(* Logix 5000 project; controller Laser_Cutter vendor 1 type 14 code 149 rev 28.11; software revision 28.00; part 3 of 4 *)
(* tags used below, declared in another part *)
   aDoorSafetySwitchUnlockSol : BOOL;
   aExhaustStart : BOOL;
   alarmActive : BOOL;
   aTapForward : BOOL;
   aTapReverse : BOOL;
   automaticSeqStep : DINT;
   autoMode : BOOL;
   autoModeReady : BOOL;
   boltDriverDownDB : TIMER;
   boltDriverUpDB : TIMER;
   boltPresentAtInfeedDB : TIMER;
   clampStation2DB : TIMER;
   clampStation4DB : TIMER;
   clampStation5DB : TIMER;
   collarAtStation1DB : TIMER;
   collarAtStation2DB : TIMER;
   collarAtStation3DB : TIMER;
   collarAtStation4DB : TIMER;
   collarAtStation5DB : TIMER;
   collarFeedingTrackHighLevelDB : TIMER;
   collarFeedingTrackLowLevelDB : TIMER;
   collarPresentAtInfeedDB : TIMER;
   Counter : DINT;
   Counter2 : DINT;
   Counter3 : DINT;
   CYCLE_IN_PROG : BOOL;
   cycleComplete : BOOL;
   doorClosedDebounceTimer : TIMER;
   doorLockedDebounceTimer : TIMER;
   doorUnlockedDebounceTimer : TIMER;
   Exec_Laser_SR : BOOL;
   Exec_Robot_SR : BOOL;
   Exec_Tapping_SR : BOOL;
   execLoadPalletSR : BOOL;
   Execute_MoveToZoneSR : BOOL;
   Execute_RejectSR : BOOL;
   executeInitializationSequence : BOOL;
   hmiMessageNumber : DINT;
   hmiMessageNumberBuffer : DINT;
   hmiMessageString : STRING;
   hmiMessageStringArray : STRING[64];
   INIT_IN_PROG : BOOL;
   initHMIMessageDelayTimer : TIMER;
   initSeqStep : DINT;
   initTimeout : TIMER;
   LaserSeqStep : INT;
   loadPalletSeqStep : INT;
   manualMode : BOOL;
   MoveToZoneSeqStep : INT;
   mSecPulseOffTmr1 : TIMER;
   mSecPulseOnTmr1 : TIMER;
   oneSecPulseOffTmr : TIMER;
   oneSecPulseOnTmr : TIMER;
   palletShotpinRetractedDebounceTimer : TIMER;
   partsPresentDurringInitialization : BOOL;
   performOpControl : CONTROL;
   performOperation : DINT[1];
   rejectPartFlag : BOOL;
   rejectSeqStep : DINT;
   rejectShuttleAtAcceptDB : TIMER;
   rejectShuttleAtRejectDB : TIMER;
   remotePVDisplayNum : DINT;
   robotAtDropAPR : BOOL;
   robotAtHome : BOOL;
   robotAtPickAPR : BOOL;
   robotFinishedDrop : BOOL;
   robotHasBolt : BOOL;
   robotInMotion : BOOL;
   robotPickBolt : BOOL;
   robotScrewInBolt : BOOL;
   robotSeqStep : DINT;
   sendRobotToDropAPR : BOOL;
   sendRobotToHome : BOOL;
   sendRobotToPick : BOOL;
   startRobotSequence : BOOL;
   systemInInitializedPosition : BOOL;
   tapDownDB : TIMER;
   tapDwellTimer : TIMER;
   tapSeqStep : DINT;
   tapUpDB : TIMER;
   unclampStation2DB : TIMER;
   unclampStation4DB : TIMER;
   unclampStation5DB : TIMER;
   walkingBeamDownDB : TIMER;
   walkingBeamLeftDB : TIMER;
   walkingBeamRightDB : TIMER;
   walkingBeamUpDB : TIMER;
   boltDriverDown : ALIAS FOR MURR_IMPACT_IO_1:I.Data[1].6;
   boltDriverUp : ALIAS FOR MURR_IMPACT_IO_1:I.Data[1].5;
   boltPresentAtInfeed : ALIAS FOR MURR_IMPACT_IO_1:I.Data[0].5;
   cameraGoodPart : ALIAS FOR Local:1:I.Data.7;
   cameraOnline : ALIAS FOR Local:1:I.Data.9;
   clampStation2 : ALIAS FOR MURR_IMPACT_IO_1:I.Data[1].7;
   clampStation4 : ALIAS FOR MURR_IMPACT_IO_1:I.Data[2].1;
   clampStation5 : ALIAS FOR MURR_IMPACT_IO_1:I.Data[2].3;
   collarAtStation1 : ALIAS FOR MURR_IMPACT_IO_1:I.Data[0].6;
   collarAtStation2 : ALIAS FOR MURR_IMPACT_IO_1:I.Data[0].7;
   collarAtStation3 : ALIAS FOR MURR_IMPACT_IO_1:I.Data[1].0;
   collarAtStation4 : ALIAS FOR MURR_IMPACT_IO_1:I.Data[1].1;
   collarAtStation5 : ALIAS FOR MURR_IMPACT_IO_1:I.Data[1].2;
   collarFeedingTrackHighLevel : ALIAS FOR MURR_IMPACT_IO_1:I.Data[0].1;
   collarFeedingTrackLowLevel : ALIAS FOR MURR_IMPACT_IO_1:I.Data[0].0;
   collarPresentAtInfeed : ALIAS FOR MURR_IMPACT_IO_1:I.Data[0].4;
   currentUser : DINT;   // Access Level of current user
   doorOpenedSafetyRelayStatus : ALIAS FOR Local:1:I.Data.1;
   doorSafetySwitchUnlockSol : ALIAS FOR Local:1:O.Data.10;
   eStopSafetyRelayStatus : ALIAS FOR Local:1:I.Data.0;
   Local1IData10 : ALIAS FOR Local:1:I.Data.10;
   Local1IData11 : ALIAS FOR Local:1:I.Data.11;
   rejectShuttleAtAccept : ALIAS FOR MURR_IMPACT_IO_1:I.Data[2].5;
   rejectShuttleAtReject : ALIAS FOR MURR_IMPACT_IO_1:I.Data[2].6;
   stopPB : ALIAS FOR Local:1:I.Data.4;
   tapDown : ALIAS FOR MURR_IMPACT_IO_1:I.Data[1].4;
   tapUp : ALIAS FOR MURR_IMPACT_IO_1:I.Data[1].3;
   TO_DRV1 : CON_EIP_IN;
   TO_DRV2 : CON_EIP_IN;
   unclampStation2 : ALIAS FOR MURR_IMPACT_IO_1:I.Data[2].0;
   unclampStation4 : ALIAS FOR MURR_IMPACT_IO_1:I.Data[2].2;
   unclampStation5 : ALIAS FOR MURR_IMPACT_IO_1:I.Data[2].4;
   walkingBeamDown : ALIAS FOR MURR_IMPACT_IO_2:I.Data[0].0;
   walkingBeamLeft : ALIAS FOR MURR_IMPACT_IO_2:I.Data[0].2;
   walkingBeamRight : ALIAS FOR MURR_IMPACT_IO_2:I.Data[0].1;
   walkingBeamUp : ALIAS FOR MURR_IMPACT_IO_1:I.Data[2].7;
(* MainProgram, continued *)

ROUTINE Exec_Reject_SR   (* ladder *)
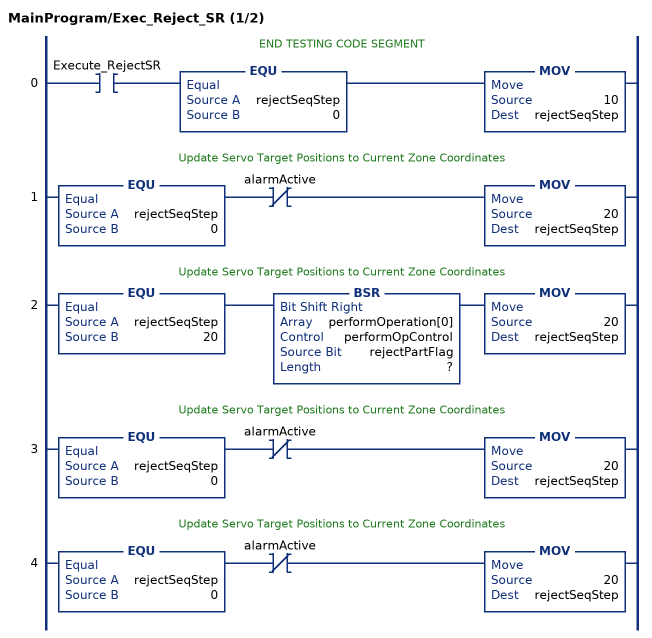
   // END TESTING CODE SEGMENT
   0: XIC(Execute_RejectSR)EQU(rejectSeqStep,0)MOV(10,rejectSeqStep);
   // Update Servo Target Positions to Current Zone Coordinates
   1: EQU(rejectSeqStep,0)XIO(alarmActive)MOV(20,rejectSeqStep);
   // Update Servo Target Positions to Current Zone Coordinates
   2: EQU(rejectSeqStep,20)BSR(performOperation[0],performOpControl,rejectPartFlag,?)MOV(20,rejectSeqStep);
   // Update Servo Target Positions to Current Zone Coordinates
   3: EQU(rejectSeqStep,0)XIO(alarmActive)MOV(20,rejectSeqStep);
   // Update Servo Target Positions to Current Zone Coordinates
   4: EQU(rejectSeqStep,0)XIO(alarmActive)MOV(20,rejectSeqStep);
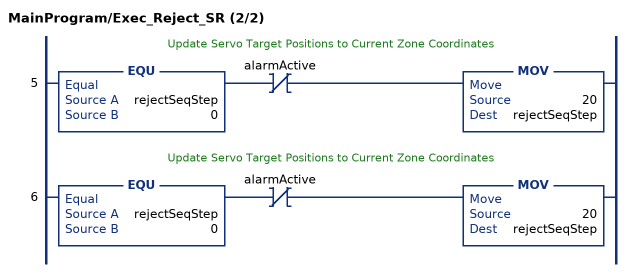
   // Update Servo Target Positions to Current Zone Coordinates
   5: EQU(rejectSeqStep,0)XIO(alarmActive)MOV(20,rejectSeqStep);
   // Update Servo Target Positions to Current Zone Coordinates
   6: EQU(rejectSeqStep,0)XIO(alarmActive)MOV(20,rejectSeqStep);
END_ROUTINE

ROUTINE Exec_Robot_SR   (* ladder *)
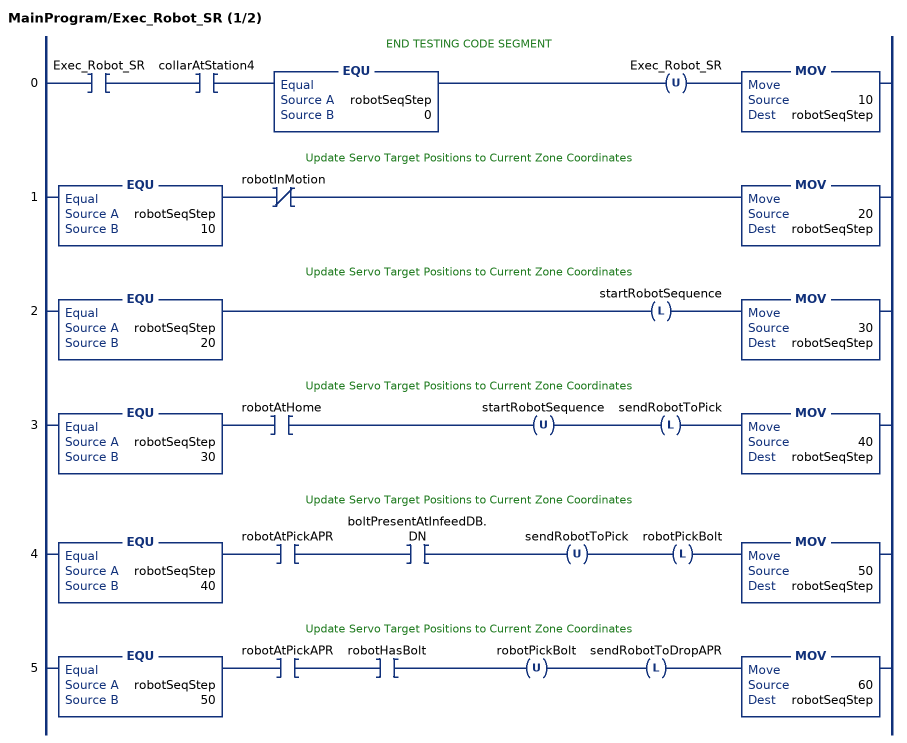
   // END TESTING CODE SEGMENT
   0: XIC(Exec_Robot_SR)XIC(collarAtStation4)EQU(robotSeqStep,0)OTU(Exec_Robot_SR)MOV(10,robotSeqStep);
   // Update Servo Target Positions to Current Zone Coordinates
   1: EQU(robotSeqStep,10)XIO(robotInMotion)MOV(20,robotSeqStep);
   // Update Servo Target Positions to Current Zone Coordinates
   2: EQU(robotSeqStep,20)OTL(startRobotSequence)MOV(30,robotSeqStep);
   // Update Servo Target Positions to Current Zone Coordinates
   3: EQU(robotSeqStep,30)XIC(robotAtHome)OTU(startRobotSequence)OTL(sendRobotToPick)MOV(40,robotSeqStep);
   // Update Servo Target Positions to Current Zone Coordinates
   4: EQU(robotSeqStep,40)XIC(robotAtPickAPR)XIC(boltPresentAtInfeedDB.DN)OTU(sendRobotToPick)OTL(robotPickBolt)MOV(50,robotSeqStep);
   // Update Servo Target Positions to Current Zone Coordinates
   5: EQU(robotSeqStep,50)XIC(robotAtPickAPR)XIC(robotHasBolt)OTU(robotPickBolt)OTL(sendRobotToDropAPR)MOV(60,robotSeqStep);
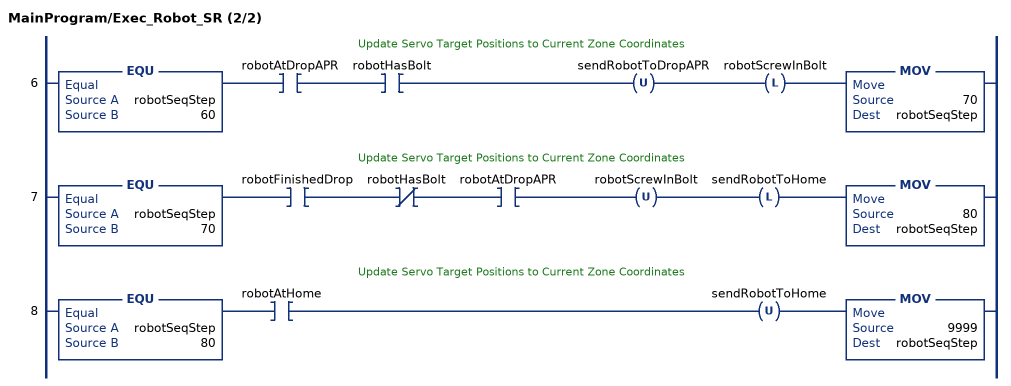
   // Update Servo Target Positions to Current Zone Coordinates
   6: EQU(robotSeqStep,60)XIC(robotAtDropAPR)XIC(robotHasBolt)OTU(sendRobotToDropAPR)OTL(robotScrewInBolt)MOV(70,robotSeqStep);
   // Update Servo Target Positions to Current Zone Coordinates
   7: EQU(robotSeqStep,70)XIC(robotFinishedDrop)XIO(robotHasBolt)XIC(robotAtDropAPR)OTU(robotScrewInBolt)OTL(sendRobotToHome)MOV(80,robotSeqStep);
   // Update Servo Target Positions to Current Zone Coordinates
   8: EQU(robotSeqStep,80)XIC(robotAtHome)OTU(sendRobotToHome)MOV(9999,robotSeqStep);
END_ROUTINE

ROUTINE Exec_Tapping_SR   (* ladder *)
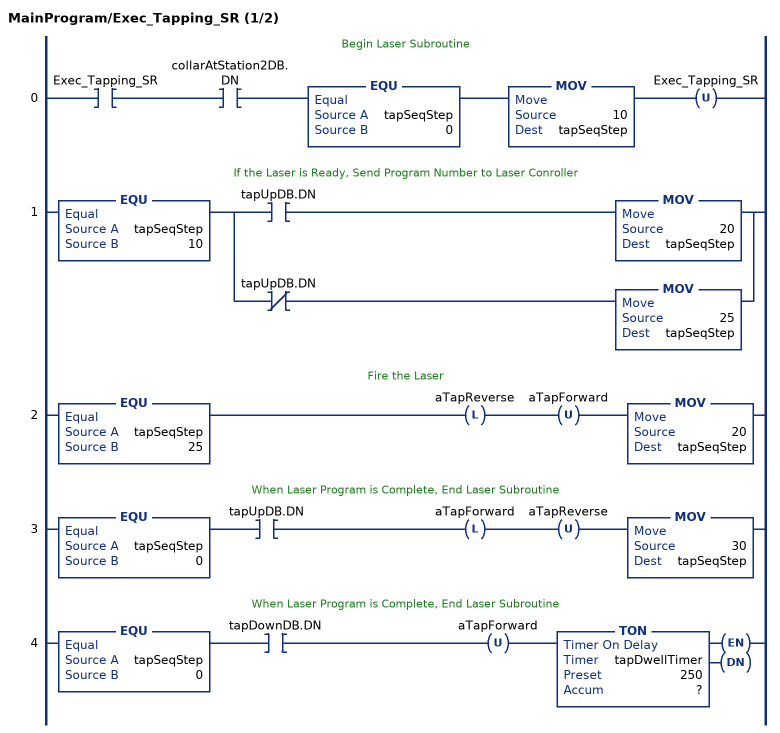
   // Begin Laser Subroutine
   0: XIC(Exec_Tapping_SR)XIC(collarAtStation2DB.DN)EQU(tapSeqStep,0)MOV(10,tapSeqStep)OTU(Exec_Tapping_SR);
   // If the Laser is Ready, Send Program Number to Laser Conroller
   1: EQU(tapSeqStep,10)[XIC(tapUpDB.DN) MOV(20,tapSeqStep) ,XIO(tapUpDB.DN) MOV(25,tapSeqStep) ];
   // Fire the Laser
   2: EQU(tapSeqStep,25)OTL(aTapReverse)OTU(aTapForward)MOV(20,tapSeqStep);
   // When Laser Program is Complete, End Laser Subroutine
   3: EQU(tapSeqStep,0)XIC(tapUpDB.DN)OTL(aTapForward)OTU(aTapReverse)MOV(30,tapSeqStep);
   // When Laser Program is Complete, End Laser Subroutine
   4: EQU(tapSeqStep,0)XIC(tapDownDB.DN)OTU(aTapForward)TON(tapDwellTimer,?,?);
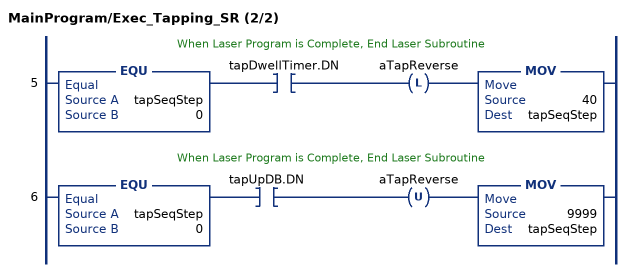
   // When Laser Program is Complete, End Laser Subroutine
   5: EQU(tapSeqStep,0)XIC(tapDwellTimer.DN)OTL(aTapReverse)MOV(40,tapSeqStep);
   // When Laser Program is Complete, End Laser Subroutine
   6: EQU(tapSeqStep,0)XIC(tapUpDB.DN)OTU(aTapReverse)MOV(9999,tapSeqStep);
END_ROUTINE

ROUTINE HMI   (* ladder *)
// HMI ROUTINE
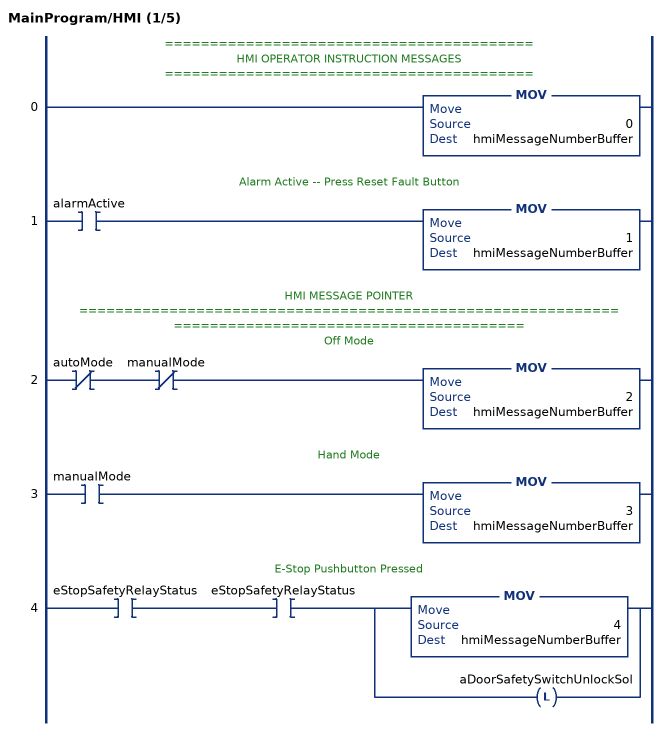
   // =========================================
   // HMI OPERATOR INSTRUCTION MESSAGES
   // =========================================
   0: MOV(0,hmiMessageNumberBuffer);
   // Alarm Active -- Press Reset Fault Button
   1: XIC(alarmActive)MOV(1,hmiMessageNumberBuffer);
   // HMI MESSAGE POINTER
   // ===================================================================================================
   // Off Mode
   2: XIO(autoMode)XIO(manualMode)MOV(2,hmiMessageNumberBuffer);
   // Hand Mode
   3: XIC(manualMode)MOV(3,hmiMessageNumberBuffer);
   // E-Stop Pushbutton Pressed
   4: XIC(eStopSafetyRelayStatus)XIC(eStopSafetyRelayStatus)[MOV(4,hmiMessageNumberBuffer) ,OTL(aDoorSafetySwitchUnlockSol) ];
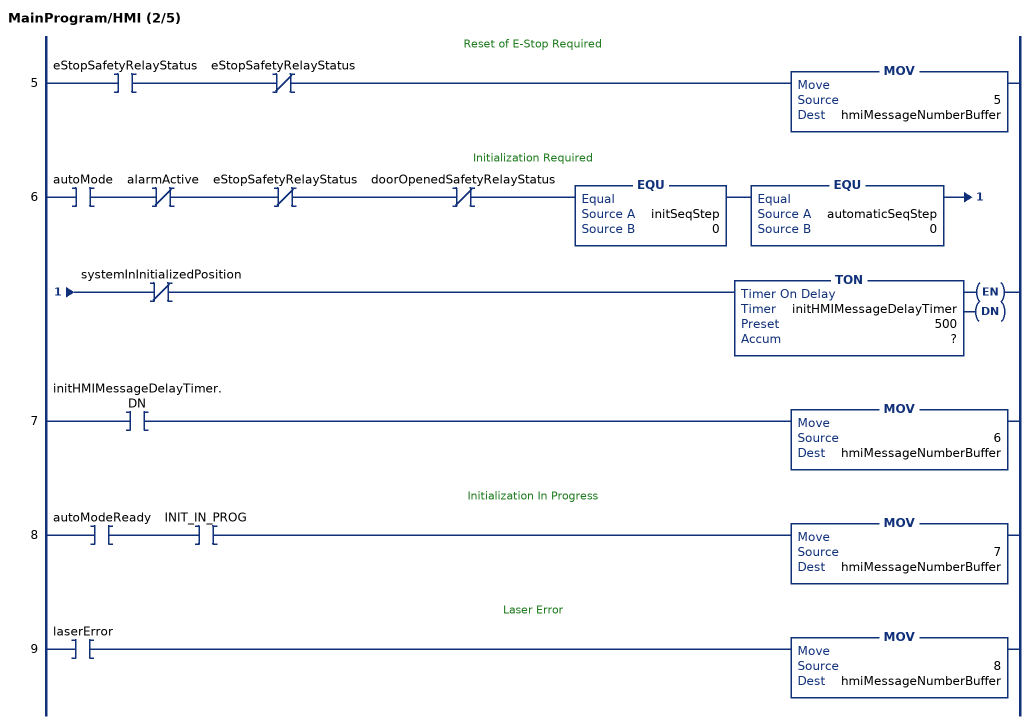
   // Reset of E-Stop Required
   5: XIC(eStopSafetyRelayStatus)XIO(eStopSafetyRelayStatus)MOV(5,hmiMessageNumberBuffer);
   // Initialization Required
   6: XIC(autoMode)XIO(alarmActive)XIO(eStopSafetyRelayStatus)XIO(doorOpenedSafetyRelayStatus)EQU(initSeqStep,0)EQU(automaticSeqStep,0)XIO(systemInInitializedPosition)TON(initHMIMessageDelayTimer,?,?);
   7: XIC(initHMIMessageDelayTimer.DN)MOV(6,hmiMessageNumberBuffer);
   // Initialization In Progress
   8: XIC(autoModeReady)XIC(INIT_IN_PROG)MOV(7,hmiMessageNumberBuffer);
   // Laser Error
   9: XIC(laserError)MOV(8,hmiMessageNumberBuffer);
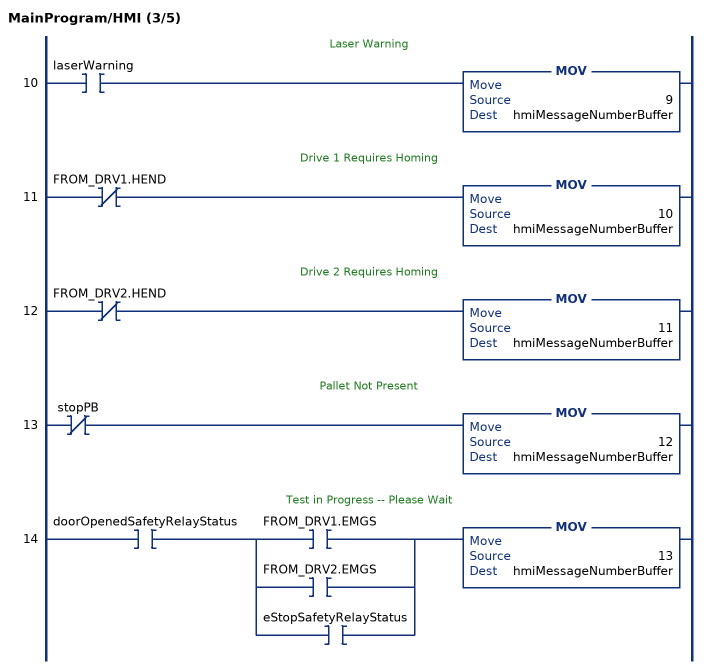
   // Laser Warning
   10: XIC(laserWarning)MOV(9,hmiMessageNumberBuffer);
   // Drive 1 Requires Homing
   11: XIO(FROM_DRV1.HEND)MOV(10,hmiMessageNumberBuffer);
   // Drive 2 Requires Homing
   12: XIO(FROM_DRV2.HEND)MOV(11,hmiMessageNumberBuffer);
   // Pallet Not Present
   13: XIO(stopPB)MOV(12,hmiMessageNumberBuffer);
   // Test in Progress -- Please Wait
   14: XIC(doorOpenedSafetyRelayStatus)[XIC(FROM_DRV1.EMGS) ,XIC(FROM_DRV2.EMGS) ,XIC(eStopSafetyRelayStatus) ]MOV(13,hmiMessageNumberBuffer);
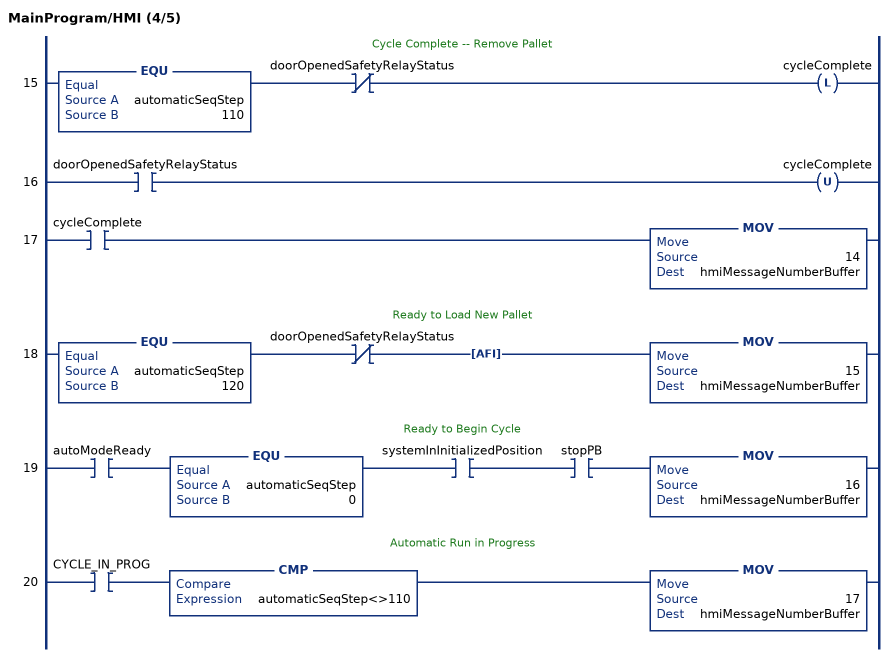
   // Cycle Complete -- Remove Pallet
   15: EQU(automaticSeqStep,110)XIO(doorOpenedSafetyRelayStatus)OTL(cycleComplete);
   16: XIC(doorOpenedSafetyRelayStatus)OTU(cycleComplete);
   17: XIC(cycleComplete)MOV(14,hmiMessageNumberBuffer);
   // Ready to Load New Pallet
   18: EQU(automaticSeqStep,120)XIO(doorOpenedSafetyRelayStatus)AFI()MOV(15,hmiMessageNumberBuffer);
   // Ready to Begin Cycle
   19: XIC(autoModeReady)EQU(automaticSeqStep,0)XIC(systemInInitializedPosition)XIC(stopPB)MOV(16,hmiMessageNumberBuffer);
   // Automatic Run in Progress
   20: XIC(CYCLE_IN_PROG)CMP(automaticSeqStep<>110)MOV(17,hmiMessageNumberBuffer);
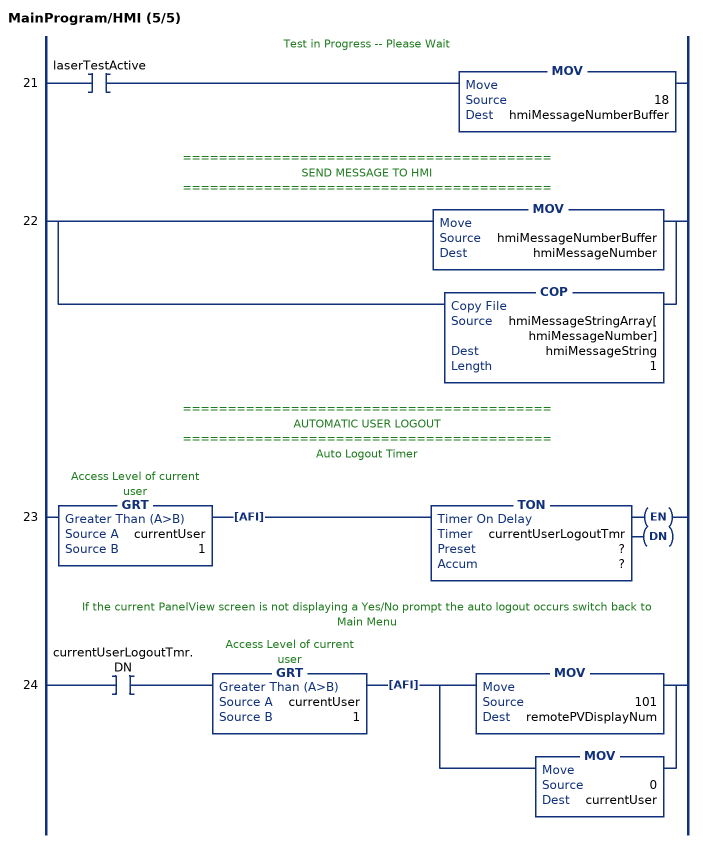
   // Test in Progress -- Please Wait
   21: XIC(laserTestActive)MOV(18,hmiMessageNumberBuffer);
   // =========================================
   // SEND MESSAGE TO HMI
   // =========================================
   22: [MOV(hmiMessageNumberBuffer,hmiMessageNumber) ,COP(hmiMessageStringArray[hmiMessageNumber],hmiMessageString,1) ];
   // =========================================
   // AUTOMATIC USER LOGOUT
   // =========================================
   // Auto Logout Timer
   23: GRT(currentUser,1)AFI()TON(currentUserLogoutTmr,?,?);
   // If the current PanelView screen is not displaying a Yes/No prompt the auto logout occurs switch back to Main Menu
   24: XIC(currentUserLogoutTmr.DN)GRT(currentUser,1)AFI()[MOV(101,remotePVDisplayNum) ,MOV(0,currentUser) ];
END_ROUTINE

ROUTINE Housekeeping   (* ladder *)
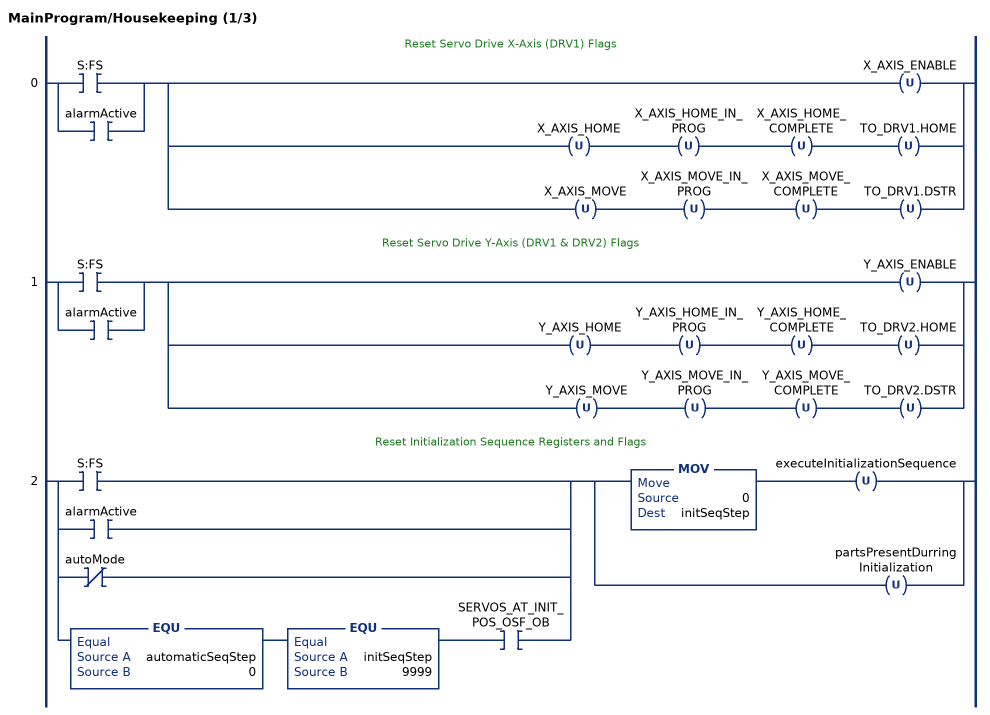
   // Reset Servo Drive X-Axis (DRV1) Flags
   0: [XIC(S:FS) ,XIC(alarmActive) ][OTU(X_AXIS_ENABLE) ,OTU(X_AXIS_HOME) OTU(X_AXIS_HOME_IN_PROG) OTU(X_AXIS_HOME_COMPLETE) OTU(TO_DRV1.HOME) ,OTU(X_AXIS_MOVE) OTU(X_AXIS_MOVE_IN_PROG) OTU(X_AXIS_MOVE_COMPLETE) OTU(TO_DRV1.DSTR) ];
   // Reset Servo Drive Y-Axis (DRV1 & DRV2) Flags
   1: [XIC(S:FS) ,XIC(alarmActive) ][OTU(Y_AXIS_ENABLE) ,OTU(Y_AXIS_HOME) OTU(Y_AXIS_HOME_IN_PROG) OTU(Y_AXIS_HOME_COMPLETE) OTU(TO_DRV2.HOME) ,OTU(Y_AXIS_MOVE) OTU(Y_AXIS_MOVE_IN_PROG) OTU(Y_AXIS_MOVE_COMPLETE) OTU(TO_DRV2.DSTR) ];
   // Reset Initialization Sequence Registers and Flags
   2: [XIC(S:FS) ,XIC(alarmActive) ,XIO(autoMode) ,EQU(automaticSeqStep,0) EQU(initSeqStep,9999) XIC(SERVOS_AT_INIT_POS_OSF_OB) ][MOV(0,initSeqStep) OTU(executeInitializationSequence) ,OTU(partsPresentDurringInitialization) ];
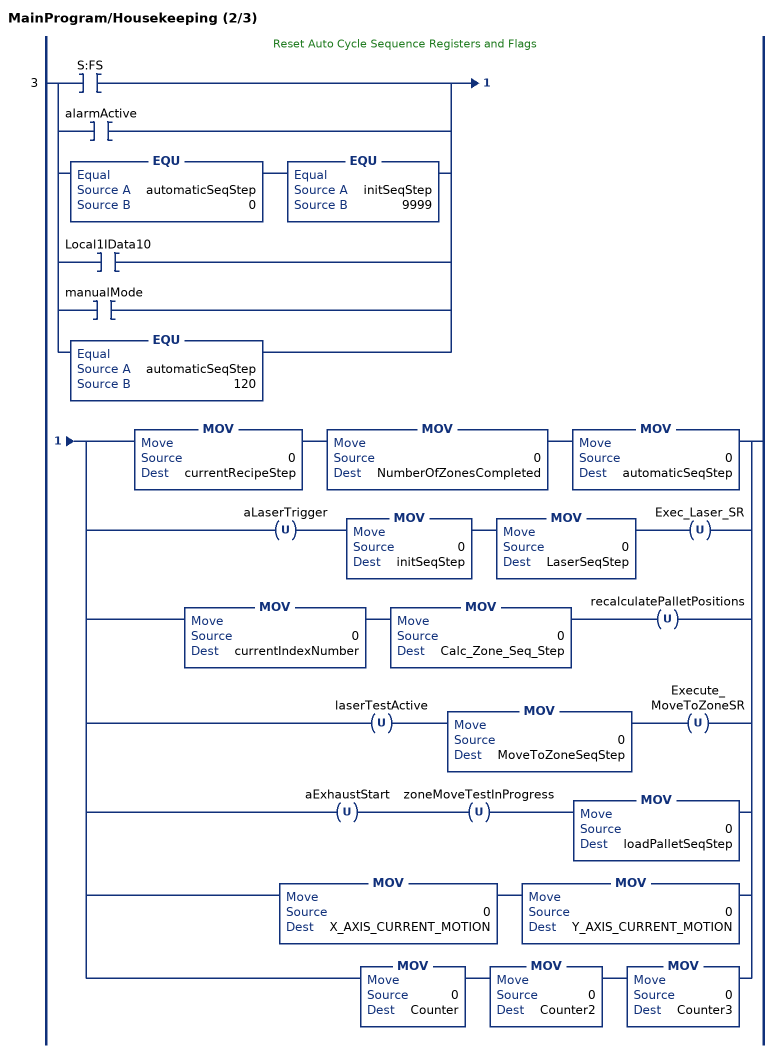
   // Reset Auto Cycle Sequence Registers and Flags
   3: [XIC(S:FS) ,[XIC(alarmActive) ,[EQU(automaticSeqStep,0) EQU(initSeqStep,9999) ,[XIC(Local1IData10) ,XIC(manualMode) ] ,EQU(automaticSeqStep,120) ] ] ][MOV(0,currentRecipeStep) MOV(0,NumberOfZonesCompleted) MOV(0,automaticSeqStep) ,OTU(aLaserTrigger) MOV(0,initSeqStep) MOV(0,LaserSeqStep) OTU(Exec_Laser_SR) ,MOV(0,currentIndexNumber) MOV(0,Calc_Zone_Seq_Step) OTU(recalculatePalletPositions) ,OTU(laserTestActive) MOV(0,MoveToZoneSeqStep) OTU(Execute_MoveToZoneSR) ,OTU(aExhaustStart) OTU(zoneMoveTestInProgress) MOV(0,loadPalletSeqStep) ,MOV(0,X_AXIS_CURRENT_MOTION) MOV(0,Y_AXIS_CURRENT_MOTION) ,MOV(0,Counter) MOV(0,Counter2) MOV(0,Counter3) ];
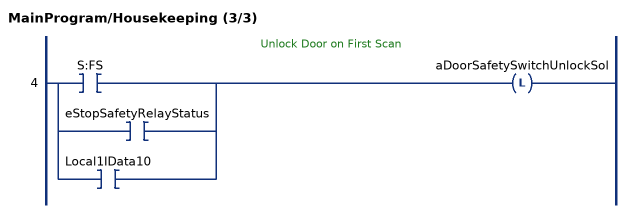
   // Unlock Door on First Scan
   4: [XIC(S:FS) ,XIC(eStopSafetyRelayStatus) ,XIC(Local1IData10) ]OTL(aDoorSafetySwitchUnlockSol);
END_ROUTINE

ROUTINE Initialization   (* ladder *)
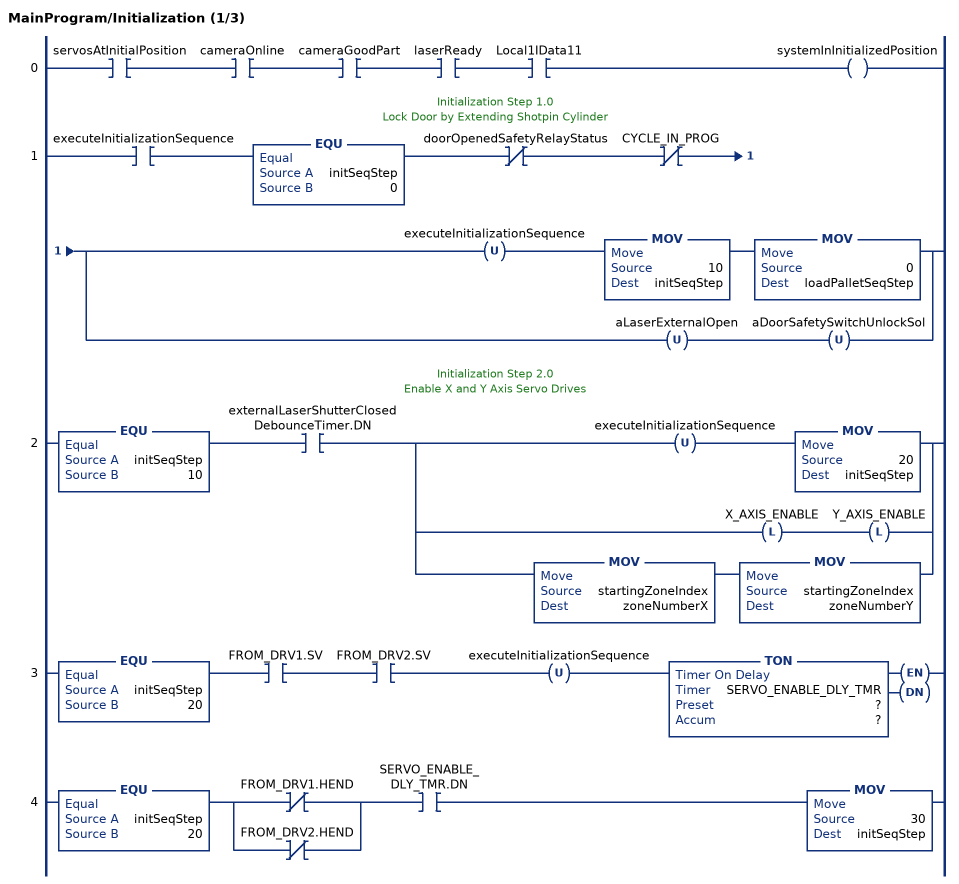
   0: XIC(servosAtInitialPosition)XIC(cameraOnline)XIC(cameraGoodPart)XIC(laserReady)XIC(Local1IData11)OTE(systemInInitializedPosition);
   // Initialization Step 1.0
   // Lock Door by Extending Shotpin Cylinder
   1: XIC(executeInitializationSequence)EQU(initSeqStep,0)XIO(doorOpenedSafetyRelayStatus)XIO(CYCLE_IN_PROG)[OTU(executeInitializationSequence) MOV(10,initSeqStep) MOV(0,loadPalletSeqStep) ,OTU(aLaserExternalOpen) OTU(aDoorSafetySwitchUnlockSol) ];
   // Initialization Step 2.0
   // Enable X and Y Axis Servo Drives
   2: EQU(initSeqStep,10)XIC(externalLaserShutterClosedDebounceTimer.DN)[OTU(executeInitializationSequence) MOV(20,initSeqStep) ,[OTL(X_AXIS_ENABLE) OTL(Y_AXIS_ENABLE) ,MOV(startingZoneIndex,zoneNumberX) MOV(startingZoneIndex,zoneNumberY) ] ];
   3: EQU(initSeqStep,20)XIC(FROM_DRV1.SV)XIC(FROM_DRV2.SV)OTU(executeInitializationSequence)TON(SERVO_ENABLE_DLY_TMR,?,?);
   4: EQU(initSeqStep,20)[XIO(FROM_DRV1.HEND) ,XIO(FROM_DRV2.HEND) ]XIC(SERVO_ENABLE_DLY_TMR.DN)MOV(30,initSeqStep);
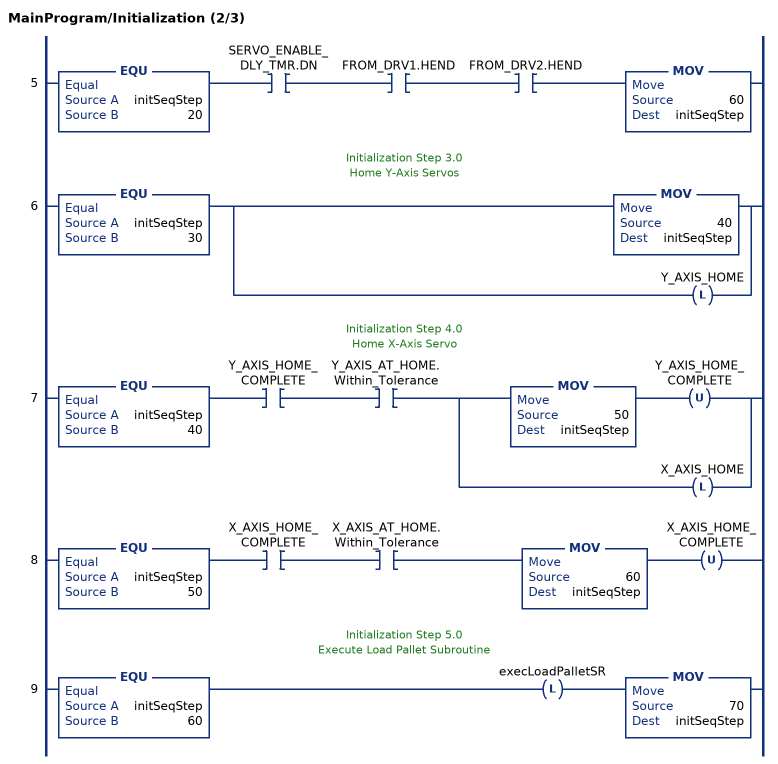
   5: EQU(initSeqStep,20)XIC(SERVO_ENABLE_DLY_TMR.DN)XIC(FROM_DRV1.HEND)XIC(FROM_DRV2.HEND)MOV(60,initSeqStep);
   // Initialization Step 3.0
   // Home Y-Axis Servos
   6: EQU(initSeqStep,30)[MOV(40,initSeqStep) ,OTL(Y_AXIS_HOME) ];
   // Initialization Step 4.0
   // Home X-Axis Servo
   7: EQU(initSeqStep,40)XIC(Y_AXIS_HOME_COMPLETE)XIC(Y_AXIS_AT_HOME.Within_Tolerance)[MOV(50,initSeqStep) OTU(Y_AXIS_HOME_COMPLETE) ,OTL(X_AXIS_HOME) ];
   8: EQU(initSeqStep,50)XIC(X_AXIS_HOME_COMPLETE)XIC(X_AXIS_AT_HOME.Within_Tolerance)MOV(60,initSeqStep)OTU(X_AXIS_HOME_COMPLETE);
   // Initialization Step 5.0
   // Execute Load Pallet Subroutine
   9: EQU(initSeqStep,60)OTL(execLoadPalletSR)MOV(70,initSeqStep);
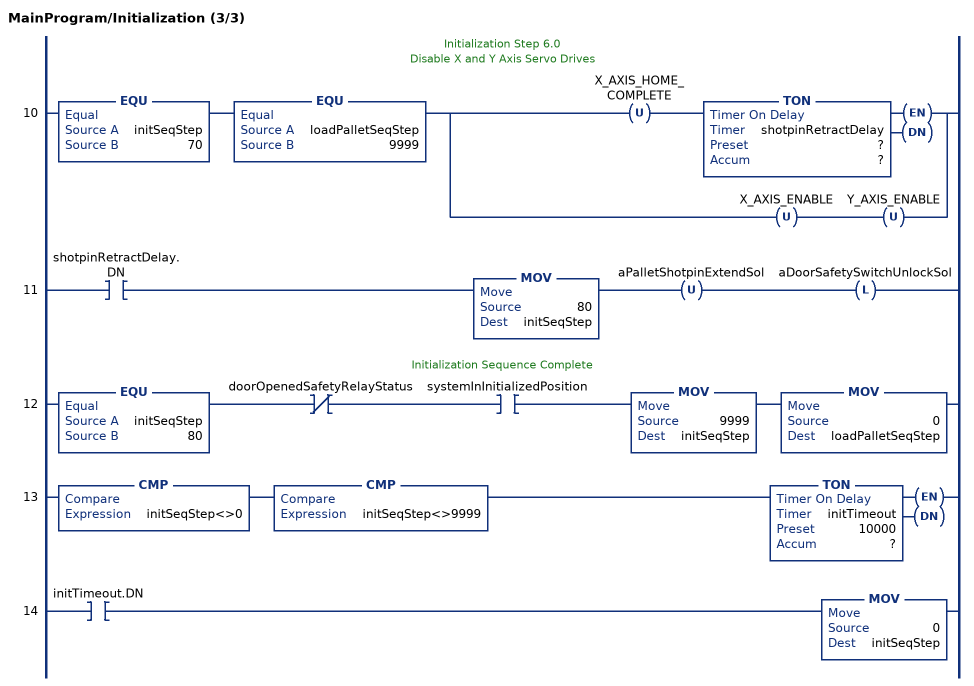
   // Initialization Step 6.0
   // Disable X and Y Axis Servo Drives
   10: EQU(initSeqStep,70)EQU(loadPalletSeqStep,9999)[OTU(X_AXIS_HOME_COMPLETE) TON(shotpinRetractDelay,?,?) ,OTU(X_AXIS_ENABLE) OTU(Y_AXIS_ENABLE) ];
   11: XIC(shotpinRetractDelay.DN)MOV(80,initSeqStep)OTU(aPalletShotpinExtendSol)OTL(aDoorSafetySwitchUnlockSol);
   // Initialization Sequence Complete
   12: EQU(initSeqStep,80)XIO(doorOpenedSafetyRelayStatus)XIC(systemInInitializedPosition)MOV(9999,initSeqStep)MOV(0,loadPalletSeqStep);
   13: CMP(initSeqStep<>0)CMP(initSeqStep<>9999)TON(initTimeout,?,?);
   14: XIC(initTimeout.DN)MOV(0,initSeqStep);
END_ROUTINE

ROUTINE Input_Debounce_Timers   (* ladder *)
// STATUS ROUTINE
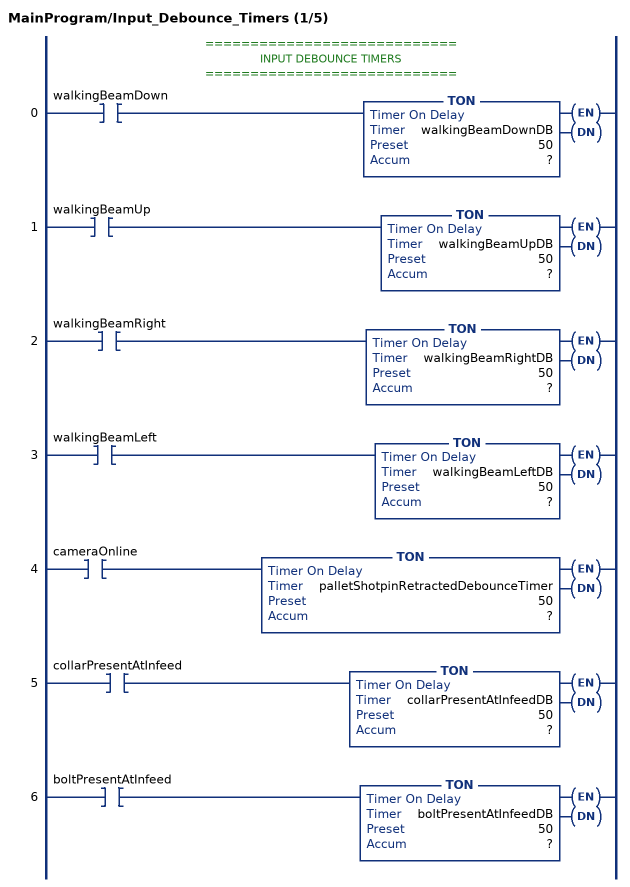
   // ============================
   // INPUT DEBOUNCE TIMERS
   // ============================
   0: XIC(walkingBeamDown)TON(walkingBeamDownDB,?,?);
   1: XIC(walkingBeamUp)TON(walkingBeamUpDB,?,?);
   2: XIC(walkingBeamRight)TON(walkingBeamRightDB,?,?);
   3: XIC(walkingBeamLeft)TON(walkingBeamLeftDB,?,?);
   4: XIC(cameraOnline)TON(palletShotpinRetractedDebounceTimer,?,?);
   5: XIC(collarPresentAtInfeed)TON(collarPresentAtInfeedDB,?,?);
   6: XIC(boltPresentAtInfeed)TON(boltPresentAtInfeedDB,?,?);
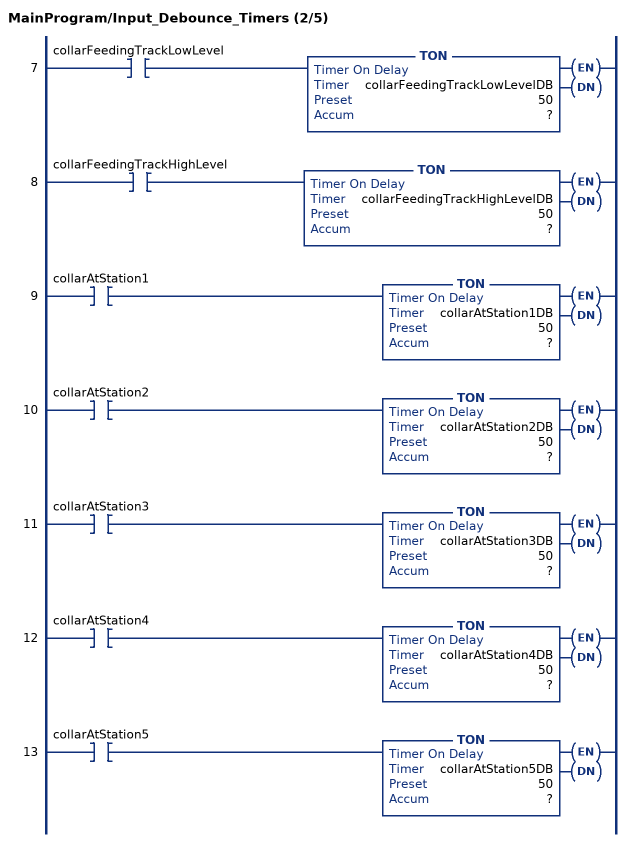
   7: XIC(collarFeedingTrackLowLevel)TON(collarFeedingTrackLowLevelDB,?,?);
   8: XIC(collarFeedingTrackHighLevel)TON(collarFeedingTrackHighLevelDB,?,?);
   9: XIC(collarAtStation1)TON(collarAtStation1DB,?,?);
   10: XIC(collarAtStation2)TON(collarAtStation2DB,?,?);
   11: XIC(collarAtStation3)TON(collarAtStation3DB,?,?);
   12: XIC(collarAtStation4)TON(collarAtStation4DB,?,?);
   13: XIC(collarAtStation5)TON(collarAtStation5DB,?,?);
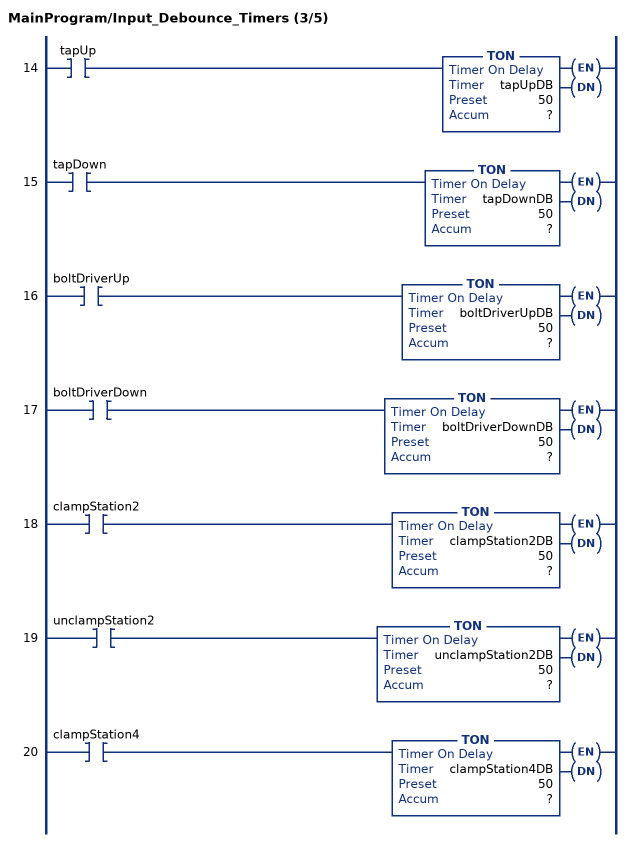
   14: XIC(tapUp)TON(tapUpDB,?,?);
   15: XIC(tapDown)TON(tapDownDB,?,?);
   16: XIC(boltDriverUp)TON(boltDriverUpDB,?,?);
   17: XIC(boltDriverDown)TON(boltDriverDownDB,?,?);
   18: XIC(clampStation2)TON(clampStation2DB,?,?);
   19: XIC(unclampStation2)TON(unclampStation2DB,?,?);
   20: XIC(clampStation4)TON(clampStation4DB,?,?);
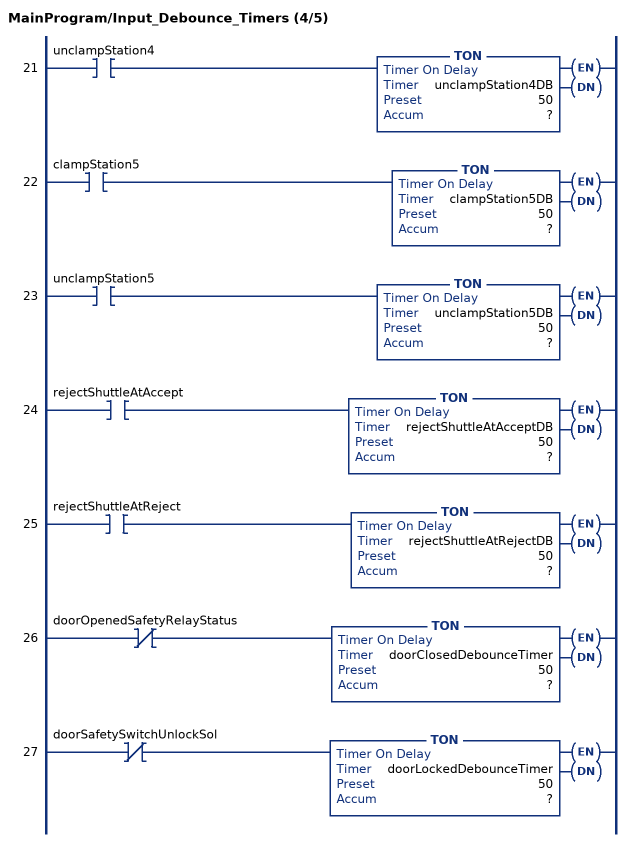
   21: XIC(unclampStation4)TON(unclampStation4DB,?,?);
   22: XIC(clampStation5)TON(clampStation5DB,?,?);
   23: XIC(unclampStation5)TON(unclampStation5DB,?,?);
   24: XIC(rejectShuttleAtAccept)TON(rejectShuttleAtAcceptDB,?,?);
   25: XIC(rejectShuttleAtReject)TON(rejectShuttleAtRejectDB,?,?);
   26: XIO(doorOpenedSafetyRelayStatus)TON(doorClosedDebounceTimer,?,?);
   27: XIO(doorSafetySwitchUnlockSol)TON(doorLockedDebounceTimer,?,?);
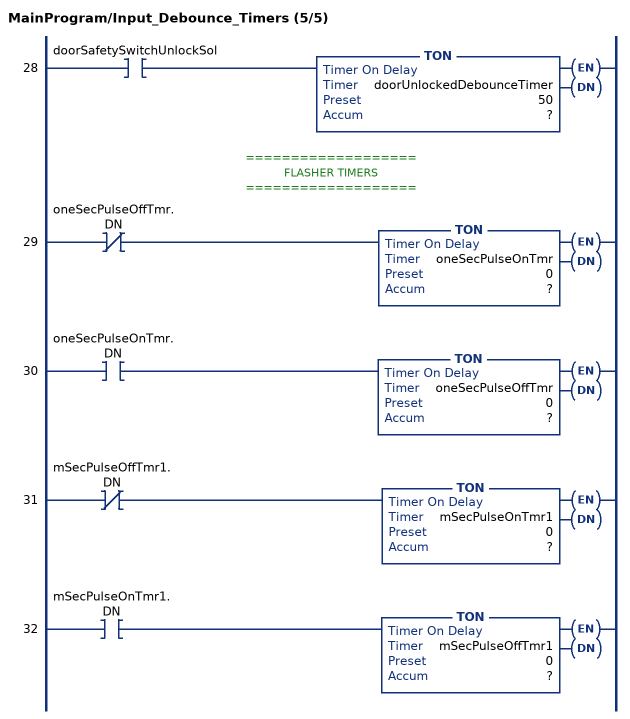
   28: XIC(doorSafetySwitchUnlockSol)TON(doorUnlockedDebounceTimer,?,?);
   // ===================
   // FLASHER TIMERS
   // ===================
   29: XIO(oneSecPulseOffTmr.DN)TON(oneSecPulseOnTmr,?,?);
   30: XIC(oneSecPulseOnTmr.DN)TON(oneSecPulseOffTmr,?,?);
   31: XIO(mSecPulseOffTmr1.DN)TON(mSecPulseOnTmr1,?,?);
   32: XIC(mSecPulseOnTmr1.DN)TON(mSecPulseOffTmr1,?,?);
END_ROUTINE
